FUNCTION_BLOCK fb_datareturn
VAR_INPUT
	dbid:UINT;
	table:STRING(50);
	start:STRING(100);
	end:STRING(100);
	bExecute:BOOL;
	
	
END_VAR
VAR_OUTPUT
	ReadStruct: ARRAY [0..1700] OF ST_ReturnedData;
	bReady:BOOL:=FALSE;
	Error:BOOL:=FALSE;
END_VAR
VAR
	sCmd:STRING(255):='';
	nstep:int:=10;
	SQLresult: FB_SQLResultEvt(sNetID:='', tTimeout:=T#5S);
	SQLcommand: FB_SQLCommandEvt(sNetid:='',tTimeout:=T#5S);
	Connectdb: FB_sqldatabaseevt(SNetID:='', tTimeout:=T#5S);
	//bExecute:BOOL:=FALSE;
	connected:BOOL:=FALSE;
	
END_VAR

	
		
IF bExecute THEN
	CASE nstep OF
	10:
				sCmd:=CONCAT('SELECT * FROM ',table);
				sCmd:=concat(sCmd, ' WHERE Dátum BETWEEN ');
				sCmd:=concat(sCmd , start);
				sCmd:=Concat(sCmd , ' AND ');
				sCmd:=concat(sCmd , end);
				sCmd:=concat(sCmd,';');
				nstep:=20;
	20:		IF connectDB.Connect(dbid) THEN
				IF connectdb.bError THEN
					Error:=TRUE;
				ELSE
					connected:=TRUE;
					nstep:=25;
				END_IF
			END_IF
		//	IF connected AND NOT connectDB.bBusy THEN 
			//	IF connectDB.CreateCmd(pSQLCommand:= ADR(SQLcommand)) THEN
			//		nstep:=30;
			//	END_IF
		//	END_IF	
		
			
	25:		IF connected THEN
				IF connectDB.CreateCmd(pSQLCommand:= ADR(SQLcommand)) THEN
					nstep:=30;
				END_IF
			END_IF						
	30:
			IF SQLcommand.ExecuteDataReturn(pSQLCmd:=ADR(sCmd),
										cbSQLCmd:=SIZEOF(sCmd),
										pSQLDBResult:=ADR(SQLResult))
			THEN
			IF sqlcommand.bError THEN
				Error:=TRUE;
			ELSE
				nstep:=40;
			END_IF
			END_IF
	40:	IF SQLResult.Read(nStartindex:= 1,
						  nRecordCount:=1001,
						  pData:=ADR(ReadStruct),
						  cbData:=SIZEOF(ReadStruct),
							TRUE, TRUE)
		THEN
		IF sqlresult.bError THEN
			Error:=TRUE;
		ELSE
			nstep:=45;
		END_IF
		END_IF	
	
	50:
		IF connectDB.Disconnect() THEN
			IF connectdb.bError THEN
				Error:=TRUE;
			ELSE
				connected:=FALSE;
				bReady:=TRUE;
				bExecute:=FALSE;	
		END_IF
		END_IF	
END_CASE
END_IF

METHOD ClearArray : BOOL
VAR_INPUT
END_VAR
memset(adr(readstruct),0,sizeof(readstruct));
END_METHOD

METHOD Reset : BOOL
VAR_INPUT
END_VAR
bReady:=FALSE;
nstep:=10;
END_METHOD

END_FUNCTION_BLOCK

(* stored: Version 1.1.0.1, ProductVersion 3.1.4024.2
   POU fb_datareturn: Id {74fe2c8c-3eed-4854-b16e-81f3686d2b76}, SpecialFunc None
   Method ClearArray: Id {99a79dab-4ac8-4bcc-9d0b-f926e5691c6f}
   Method Reset: Id {3451f12f-e189-4ec8-a629-804e9a81d2d9} *)
